TYPE ST_HmiEventJson :
STRUCT
	eplan				: STRING;
	popUp				: BOOL;
END_STRUCT
END_TYPE

(* stored: Version 1.1.0.1
   DUT ST_HmiEventJson: Id {d059d8e6-1265-429e-829d-93f6fd693400} *)
